// TIA Portal project "PNP_SENSOR_CONNECTION" (V15)

(* hardware
DEVICE "S7-1200 station_1"  S7-1200 Station
   slot 0: "Rack_0"  S7-1200 Rack  Rack  V1.0
   slot 1: "PLC_1"  CPU 1212C DC/DC/DC  6ES7 212-1AD30-0XB0  V2.2
*)

// ===== PLC "PLC_1"  CPU 1212C DC/DC/DC =====

VAR_GLOBAL   // PLC tag table "Default tag table"
   "I_ESTOP" AT %I0.0 : Bool;   // ACIL STOP BUTONU
   "I_START_BTN" AT %I0.1 : Bool;   // START BUTONU
   "I_STOP_BTN" AT %I0.2 : Bool;   // STOP BUTONU
   "I_THERMAL_RELAY" AT %I0.3 : Bool;   // TERMIK ROLE
   "I_MOTOR_PROJECTION" AT %I0.4 : Bool;   // MOTOR KORUMA ROLESI
   "I_LIMIT_SWITCH" AT %I0.5 : Bool;   // SINIR ANAHTARI
   "I_INDUCTIVE_SENSOR" AT %I0.6 : Bool;   // ENDUKTIF SENSOR
   "I_OPTICAL_SENSOR" AT %I0.7 : Bool;   // OPTIK SENSOR
   "Q_RELAY_1" AT %Q0.0 : Bool;   // RÖLE 1
   "Q_RELAY_2" AT %Q0.1 : Bool;   // RÖLE 2
   "Q_RELAY_3" AT %Q0.2 : Bool;   // RÖLE 3
   "Q_RELAY_4" AT %Q0.3 : Bool;   // RÖLE 4
   "Q_RELAY_5" AT %Q0.4 : Bool;   // RÖLE 5
   "Q_RELAY_6" AT %Q0.5 : Bool;   // RÖLE 6
END_VAR

ORGANIZATION_BLOCK "Main"   // OB1, LAD, ProgramCycle
TITLE = "Main Program Sweep (Cycle)"
{ S7_Optimized_Access := 'TRUE' }
VERSION : 0.1
BEGIN

REGION Network 1: RÖLE 1
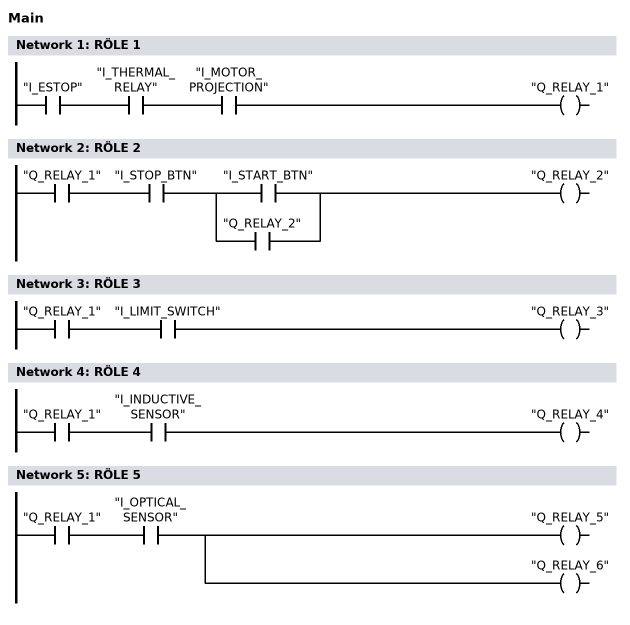
   RUNG wire#powerrail
      Contact( "I_ESTOP" )
      Contact( "I_THERMAL_RELAY" )
      Contact( "I_MOTOR_PROJECTION" )
      Coil( "Q_RELAY_1" )
   END_RUNG
   // the same network as SCL:
   "Q_RELAY_1" := "I_ESTOP" AND "I_THERMAL_RELAY" AND "I_MOTOR_PROJECTION";
END_REGION

REGION Network 2: RÖLE 2
   RUNG wire#powerrail
      Contact( "Q_RELAY_1" )
      Contact( "I_STOP_BTN" )
      wire#w1
      Contact( "I_START_BTN" )
      wire#w2
      Coil( "Q_RELAY_2" )
   END_RUNG
   RUNG wire#w1
      Contact( "Q_RELAY_2" )
   END_RUNG wire#w2
   // the same network as SCL:
   "Q_RELAY_2" := "Q_RELAY_1" AND "I_STOP_BTN" AND ("I_START_BTN" OR "Q_RELAY_2");
END_REGION

REGION Network 3: RÖLE 3
   RUNG wire#powerrail
      Contact( "Q_RELAY_1" )
      Contact( "I_LIMIT_SWITCH" )
      Coil( "Q_RELAY_3" )
   END_RUNG
   // the same network as SCL:
   "Q_RELAY_3" := "Q_RELAY_1" AND "I_LIMIT_SWITCH";
END_REGION

REGION Network 4: RÖLE 4
   RUNG wire#powerrail
      Contact( "Q_RELAY_1" )
      Contact( "I_INDUCTIVE_SENSOR" )
      Coil( "Q_RELAY_4" )
   END_RUNG
   // the same network as SCL:
   "Q_RELAY_4" := "Q_RELAY_1" AND "I_INDUCTIVE_SENSOR";
END_REGION

REGION Network 5: RÖLE 5
   RUNG wire#powerrail
      Contact( "Q_RELAY_1" )
      Contact( "I_OPTICAL_SENSOR" )
      wire#w1
      Coil( "Q_RELAY_5" )
   END_RUNG
   RUNG wire#w1
      Coil( "Q_RELAY_6" )
   END_RUNG
   // the same network as SCL:
   "Q_RELAY_5" := "Q_RELAY_1" AND "I_OPTICAL_SENSOR";
   "Q_RELAY_6" := "Q_RELAY_5";
END_REGION
END_ORGANIZATION_BLOCK